PROGRAM MAIN
VAR
		
		
		

END_VAR

// Init
Init_Devices();
//
Get_PID_Gain();


GVL.AxisX_Power_Fuc.Enable := GVL.OnMoterX;
GVL.AxisY_Power_Fuc.Enable := GVL.OnMoterY;



GVL.AxisX_AbMove_Fuc.Execute := GVL.X_AbMove_Ex;
GVL.X_AbMove_Ex := FALSE;


GVL.AxisY_AbMove_Fuc.Execute := GVL.Y_AbMove_Ex;
GVL.Y_AbMove_Ex := FALSE;


GVL.fbCoEWrite_X(
		Axis :=GVL.AxisX,		
		NetId := '5.33.182.40.1.1', 
  		Index := GVL.Index,
  		pSrcBuf := ADR(GVL.X_Gain), 
  		BufLen := SIZEOF(GVL.X_Gain), 
  		Execute := GVL.X_COE_Ex, 
  		Timeout := T#1S, 	
		CompleteAccess := GVL.CompleteAccess, 
		Busy => GVL.Success
	);	
	
GVL.fbCoEWrite_Y(
		Axis :=GVL.AxisY,		
		NetId := '5.33.182.40.1.1', 
  		Index := GVL.Index,
  		pSrcBuf := ADR(GVL.Y_Gain), 
  		BufLen := SIZEOF(GVL.Y_Gain), 
  		Execute := GVL.Y_COE_Ex, 
  		Timeout := T#1S, 	
		CompleteAccess := GVL.CompleteAccess, 
		Busy => GVL.Success
	);

END_PROGRAM

(* stored: Version 1.1.0.1, ProductVersion 3.1.4024.12
   POU MAIN: Id {4fff3968-6d8d-4583-a644-d7c373040352}, SpecialFunc None *)
